{attribute 'qualified_only'}
VAR_GLOBAL
	sET	:	STRING := 'ABC';
END_VAR

(* stored: Version 1.1.0.1
   GVL GVL_SIM: Id {18ec3a91-aef1-0987-253b-bb587281437a} *)
